// TIA Portal V16 export
// export: Created 2021-11-12T13:31:02.2452231Z, ExportSetting WithDefaults, DisplayName Totally Integrated Automation Portal, DisplayVersion V16 Update 3, DisplayName TIA Portal Version Control Interface, DisplayVersion V16 Update 2, DisplayName TIA Portal Openness, DisplayVersion V16 Update 3, DisplayName SINAMICS Startdrive Advanced, DisplayVersion V16 Update 5, DisplayName SINAMICS Startdrive G130, G150, S120, S150, SINAMICS MV, S210, DisplayVersion V16 Update 5, DisplayName SINAMICS Startdrive G110M, G120, G120C, G120D, G120P, G115D, DisplayVersion V16 Update 5, DisplayName STEP 7 Professional, DisplayVersion V16 Update 3, DisplayName STEP 7 Safety, DisplayVersion V16, DisplayName WinCC UA Professional, DisplayVersion V16 Update 3
DATA_BLOCK "IDB_Safety_Aux"   // DB192
{ DB_Accessible_From_OPC_UA := 'FALSE' }
VERSION : 0.1
// stored: AutoNumber true, DBAccessibleFromOPCUA false, InstanceOfName Safety_Aux, InstanceOfType FB
"Safety_Aux"
   // VAR
   //    "SF_100+RU01-QQ01" : "STD_EuchnerDoor";
   //    "SF_100+RU01-QQ02" { S7_SetPoint := 'True'} : "STD_EuchnerDoor";
   //    "SF_100+RU01-QQ03" { S7_SetPoint := 'True'} : "STD_EuchnerDoor";
   //    "SF_100+RU01-QQ04" { S7_SetPoint := 'True'} : "STD_EuchnerDoor";
   //    "SF_100+RU01-QQ05" { S7_SetPoint := 'True'} : "STD_EuchnerDoor";
   //    "SF_100+RU01-QQ06" { S7_SetPoint := 'True'} : "STD_EuchnerDoor";
   //    "SF_100+RU01-QQ07" { S7_SetPoint := 'True'} : "STD_EuchnerDoor";
   //    "SF_100+RU01-QQ08" { S7_SetPoint := 'True'} : "STD_EuchnerDoor";
   //    "SF_200+RU01-QQ01" { S7_SetPoint := 'True'} : "STD_EuchnerDoor";
   //    "SF_200+RU01-QQ02" { S7_SetPoint := 'True'} : "STD_EuchnerDoor";
   //    "SF_200+RU01-QQ03" { S7_SetPoint := 'True'} : "STD_EuchnerDoor";
   //    "SF_200+RU01-QQ04" { S7_SetPoint := 'True'} : "STD_EuchnerDoor";
   //    "SF_200+RU01-QQ05" { S7_SetPoint := 'True'} : "STD_EuchnerDoor";
   //    "SF_100+RU01-KF01" { S7_SetPoint := 'True'} : "STD_EuchnerSafetySwitch2MBM";
   //    "SF_100+RU01-KF02" { S7_SetPoint := 'True'} : "STD_EuchnerSafetySwitch2MBM";
   //    "SF_100+RU01-KF03" { S7_SetPoint := 'True'} : "STD_EuchnerSafetySwitch2MBM";
   //    "SF_200+RU01-KF01" { S7_SetPoint := 'True'} : "STD_EuchnerSafetySwitch2MBM";
   //    "SF_200+RU01-KF02" { S7_SetPoint := 'True'} : "STD_EuchnerSafetySwitch2MBM";
   //    "SF_200+RU01-KF03" { S7_SetPoint := 'True'} : "STD_EuchnerSafetySwitch2MBM";
   //    "SF_200+RU01-KF04" { S7_SetPoint := 'True'} : "STD_EuchnerSafetySwitch2MBM";
   //    SF_KAS1_ES { S7_SetPoint := 'True'} : "STD_DI_Mon";
   //    SF_KAS2_ES { S7_SetPoint := 'True'} : "STD_DI_Mon";
   //    SF_BSN1_2_ES { S7_SetPoint := 'True'} : "STD_DI_Mon";
   //    SF_BSN3_ES { S7_SetPoint := 'True'} : "STD_DI_Mon";
   //    SF_BSN4_5_ES { S7_SetPoint := 'True'} : "STD_DI_Mon";
   //    SF_SCH1_ES { S7_SetPoint := 'True'} : "STD_DI_Mon";
   //    SF_THM1_ES { S7_SetPoint := 'True'} : "STD_DI_Mon";
   //    SF_THM2_ES { S7_SetPoint := 'True'} : "STD_DI_Mon";
   //    "SF_000UH10-SF01_ES" { S7_SetPoint := 'True'} : "STD_DI_Mon";
   //    "SF_000UH11-SF01_ES" { S7_SetPoint := 'True'} : "STD_DI_Mon";
   //    "SF_100UH11-SF01_ES" { S7_SetPoint := 'True'} : "STD_DI_Mon";
   //    "SF_100UH12-SF01_ES" { S7_SetPoint := 'True'} : "STD_DI_Mon";
   //    "SF_100UH13-SF01_ES" { S7_SetPoint := 'True'} : "STD_DI_Mon";
   //    "SF_100UF01-SF01_ES" { S7_SetPoint := 'True'} : "STD_DI_Mon";
   //    "SF_200UH11-SF01_ES" { S7_SetPoint := 'True'} : "STD_DI_Mon";
   //    "SF_210UF01-SF01_ES" { S7_SetPoint := 'True'} : "STD_DI_Mon";
   //    "SF_220UF01-SF01_ES" { S7_SetPoint := 'True'} : "STD_DI_Mon";
   //    "SF_230UF01-SF01_ES" { S7_SetPoint := 'True'} : "STD_DI_Mon";
   //    "SF_200UF01-SF01_ES" { S7_SetPoint := 'True'} : "STD_DI_Mon";
   //    "SF_300UH11-SF01_ES" { S7_SetPoint := 'True'} : "STD_DI_Mon";
   //    "SF_310UH31-SF01_ES" { S7_SetPoint := 'True'} : "STD_DI_Mon";
   //    "SF_330UF01-SF01_ES" { S7_SetPoint := 'True'} : "STD_DI_Mon";
   //    "SF_400UH11-SF01_ES" { S7_SetPoint := 'True'} : "STD_DI_Mon";
   //    "SF_410UH31-SF01_ES" { S7_SetPoint := 'True'} : "STD_DI_Mon";
   //    "SF_420UH31-SF01_ES" { S7_SetPoint := 'True'} : "STD_DI_Mon";
   //    "SF_430UF01-SF01_ES" { S7_SetPoint := 'True'} : "STD_DI_Mon";
   //    SF_100QQ01_ES { S7_SetPoint := 'True'} : "STD_DI_Mon";
   //    SF_100QQ02_ES { S7_SetPoint := 'True'} : "STD_DI_Mon";
   //    SF_100QQ03_ES { S7_SetPoint := 'True'} : "STD_DI_Mon";
   //    SF_100QQ04_ES { S7_SetPoint := 'True'} : "STD_DI_Mon";
   //    SF_100QQ05_ES { S7_SetPoint := 'True'} : "STD_DI_Mon";
   //    SF_100QQ06_ES { S7_SetPoint := 'True'} : "STD_DI_Mon";
   //    SF_100QQ07_ES { S7_SetPoint := 'True'} : "STD_DI_Mon";
   //    SF_100QQ08_ES { S7_SetPoint := 'True'} : "STD_DI_Mon";
   //    SF_200QQ01_ES { S7_SetPoint := 'True'} : "STD_DI_Mon";
   //    SF_200QQ02_ES { S7_SetPoint := 'True'} : "STD_DI_Mon";
   //    SF_200QQ03_ES { S7_SetPoint := 'True'} : "STD_DI_Mon";
   //    SF_200QQ04_ES { S7_SetPoint := 'True'} : "STD_DI_Mon";
   //    SF_200QQ05_ES { S7_SetPoint := 'True'} : "STD_DI_Mon";
   //    SF_1R1RC01_ES { S7_SetPoint := 'True'} : "STD_DI_Mon";
   //    SF_1R2RC01_ES { S7_SetPoint := 'True'} : "STD_DI_Mon";
   //    SF_1R3RC01_ES { S7_SetPoint := 'True'} : "STD_DI_Mon";
   //    SF_1R4RC01_ES { S7_SetPoint := 'True'} : "STD_DI_Mon";
   //    SF_1R5RC01_ES { S7_SetPoint := 'True'} : "STD_DI_Mon";
   //    SF_1R6RC01_ES { S7_SetPoint := 'True'} : "STD_DI_Mon";
   //    SF_2R1RC01_ES { S7_SetPoint := 'True'} : "STD_DI_Mon";
   //    SF_2R2RC01_ES { S7_SetPoint := 'True'} : "STD_DI_Mon";
   //    "SF_000UH01-KF31" { S7_SetPoint := 'True'} : "STD_DI_Mon";
   //    "SF_000UH01-KF32" { S7_SetPoint := 'True'} : "STD_DI_Mon";
   //    "SF_000UH01-KF33" { S7_SetPoint := 'True'} : "STD_DI_Mon";
   //    "SF_000UH01-KF41" { S7_SetPoint := 'True'} : "STD_DI_Mon";
   //    "SF_000UH11-KF31" { S7_SetPoint := 'True'} : "STD_DI_Mon";
   //    "SF_000UH11-KF32" { S7_SetPoint := 'True'} : "STD_DI_Mon";
   //    "SF_100UH11-KF31" { S7_SetPoint := 'True'} : "STD_DI_Mon";
   //    "SF_100UH12-KF31" { S7_SetPoint := 'True'} : "STD_DI_Mon";
   //    "SF_100UH13-KF31" { S7_SetPoint := 'True'} : "STD_DI_Mon";
   //    "SF_100UH13-KF32" { S7_SetPoint := 'True'} : "STD_DI_Mon";
   //    "SF_200UH11-KF31" { S7_SetPoint := 'True'} : "STD_DI_Mon";
   //    "SF_300UH11-KF31" { S7_SetPoint := 'True'} : "STD_DI_Mon";
   //    "SF_310UH31-KF31" { S7_SetPoint := 'True'} : "STD_DI_Mon";
   //    "SF_400UH11-KF31" { S7_SetPoint := 'True'} : "STD_DI_Mon";
   //    "SF_410UH31-KF31" { S7_SetPoint := 'True'} : "STD_DI_Mon";
   //    "SF_420UH31-KF31" { S7_SetPoint := 'True'} : "STD_DI_Mon";
   //    "SF_100RU01-KF01" { S7_SetPoint := 'True'} : "STD_DI_Mon";
   //    "SF_100RU01-KF02" { S7_SetPoint := 'True'} : "STD_DI_Mon";
   //    "SF_100RU01-KF03" { S7_SetPoint := 'True'} : "STD_DI_Mon";
   //    "SF_200RU01-KF01" { S7_SetPoint := 'True'} : "STD_DI_Mon";
   //    "SF_200RU01-KF02" { S7_SetPoint := 'True'} : "STD_DI_Mon";
   //    "SF_200RU01-KF03" { S7_SetPoint := 'True'} : "STD_DI_Mon";
   //    "SF_200RU01-KF04" { S7_SetPoint := 'True'} : "STD_DI_Mon";
   // END_VAR
BEGIN
END_DATA_BLOCK
